(* CODESYS project Thermoversuch_00_20.project
   Description: Receives some incoming messages and echoes them with CAN-ID +1
   Company: 3S - Smart Software Solutions GmbH
   Version: 1.0.0.0
   Title: CAN Bus API Example
   Author: 3S - Smart Software Solutions GmbH

Project tree, tasks and I/O mapping:
  XLH : CODESYS Control for Raspberry Pi 64 SL, CODESYS, order no. 2302000009, version 4.12.0.0
    application app
      libraries: CAN API, 1.0.0.3 (3S - Smart Software Solutions GmbH); Standard, 3.5.18.0 (System); Memory, * (3S - Smart Software Solutions GmbH); Util, 3.5.19.0 (System); VisuDialogs, * (System); CAA Tick Extern, 3.5.17.0 (CAA Technical Workgroup); SysTime, 3.5.17.0 (System); CmpIecTask, * (System); xemax Bibliothek, 0.20 (xemax ag)
      task MAIN_TASK (cyclic, interval 20 ms, priority 0) calls MAIN, io
      task VISU_TASK (cyclic, interval 100 ms, priority 31) calls VisuElems.Visu_Prg
      program io [ST]
      Symbols
      visualisation Visualization
      program MAIN [ST]: CALL_CFC
      RNDIS_Driver
    SoftMotion General Axis Pool
    GPIOs_A_B : GPIOs B+/Pi2, CODESYS, version 4.12.0.0
        input  app.io.bSw1 : BOOL  // digital inputs (GPIO0..GPIO31).Bit4
        input  app.io.bSw2 : BOOL  // digital inputs (GPIO0..GPIO31).Bit5
        input  app.io.bSw3 : BOOL  // digital inputs (GPIO0..GPIO31).Bit6
        input  app.io.bSw4 : BOOL  // digital inputs (GPIO0..GPIO31).Bit12
        input  app.io.bSw5 : BOOL  // digital inputs (GPIO0..GPIO31).Bit13
        input  app.io.bSw6 : BOOL  // digital inputs (GPIO0..GPIO31).Bit16
        input  app.io.bSw7 : BOOL  // digital inputs (GPIO0..GPIO31).Bit17
        input  app.io.bSw8 : BOOL  // digital inputs (GPIO0..GPIO31).Bit19
        output app.io.bLed1 : BOOL  // digital outputs (GPIO0..GPIO31).Bit20
        output app.io.bLed2 : BOOL  // digital outputs (GPIO0..GPIO31).Bit21
        output app.io.bLed3 : BOOL  // digital outputs (GPIO0..GPIO31).Bit22
        output app.io.bLed4 : BOOL  // digital outputs (GPIO0..GPIO31).Bit23
        output app.io.bLed5 : BOOL  // digital outputs (GPIO0..GPIO31).Bit24
        output app.io.bLed6 : BOOL  // digital outputs (GPIO0..GPIO31).Bit26
        output app.io.bLed7 : BOOL  // digital outputs (GPIO0..GPIO31).Bit27
        unmapped channels: digital inputs (GPIO0..GPIO31), digital outputs (GPIO0..GPIO31)
    Onewire
    Camera device
      <Leer>
    SPI
    I²C
    Ethernet : Ethernet, CODESYS, version 4.2.0.0
        settings: IPAddress = [127,0,0,1]; SubnetMask = [255,0,0,0]; GatewayAddress = [0,0,0,0]; NetworkInterfaceName = 'lo'; NetworkInterfaceName = "lo"; SaveCommunicationSettings = FALSE
      ModbusTCP_Slave_OLED_Port_503 : ModbusTCP Slave Device, CODESYS, version 4.3.0.0
          settings: Port = 503
          output app.io.oled.awToOled : ARRAY[0..32] OF WORD  // Ausgänge
          unmapped channels: Eingänge
  libraries: VisuSymbols, 4.5.0.0 (System); DepictorBase, 1.0.5.0 (3S - Smart Software Solutions GmbH)
  text list GlobalTextList
  00000000-0000-0000-0000-000000000000|E:\xemax ag\prj_24_03_xLH - Allgemein\Image\RNDIS_Driver.zip
*)

// XLH/app/MAIN
PROGRAM MAIN
VAR
	bStartup: BOOL := TRUE;
	rDummy: REAL;
	bDummy: BOOL;
	data_logger: DATA_LOGGER;
	iXyDiagrammMin: INT;
	iXyDiagrammMax: INT;
	iXyDiagrammMaxVisu: INT;
	sLoggerBuffer: STRING(255);
	bRelaisVisu: BOOL;
	vVersionPlc: VERSION;
	sVersionPlc: STRING(255);
	vVersionLib: VERSION;
	sVersionLib: STRING(255);
END_VAR

// Version Bibliothex xemax
vVersionPlc.uiMajor := 0;
vVersionPlc.uiMinor := 10;
sVersionPlc := CONCAT(TO_STRING(TO_UINT(vVersionPlc.uiMajor)), CONCAT('.', (TO_STRING(TO_UINT(vVersionPlc.uiMinor)))));
vVersionLib := xemax.GetLibVersion();
sVersionLib := CONCAT(TO_STRING(TO_UINT(vVersionLib.uiMajor)), CONCAT('.', (TO_STRING(TO_UINT(vVersionLib.uiMinor)))));

IF bStartup THEN
	bStartup := FALSE;
	io.shelly.sIpShelly := '192.168.1.51';
END_IF

// Maximaler Index der Visualisierung
iXyDiagrammMax := data_logger.iIndexMax - iXyDiagrammMaxVisu;
// Status des Datenloggers
sLoggerBuffer := TO_STRING(TO_INT(MAIN.data_logger.rTimeSinceStart));
sLoggerBuffer := CONCAT(sLoggerBuffer, 's / ');
sLoggerBuffer := CONCAT(sLoggerBuffer, TO_STRING(TO_INT(data_logger.iIndexMax)));
sLoggerBuffer := CONCAT(sLoggerBuffer, 's');

bDummy := io.shelly.bRelais;
bDummy := io.shelly.bRelaisState;

rDummy := io.shelly.rVoltage;
rDummy := io.shelly.rCurrent;
rDummy := io.shelly.rActivePower;

rDummy := io.shelly.rTemperature1;
rDummy := io.shelly.rTemperature2;
rDummy := io.shelly.rTemperature3;

io.bLed1 := io.bSw1;
io.bLed2 := io.bSw2;
io.bLed3 := io.bSw3;
io.bLed4 := io.bSw4;
io.bLed5 := io.bSw5;
io.bLed6 := io.bSw6;
io.bLed7 := io.bSw7;

io.oled.bShowLines := io.bSw8;
io.oled.sLine1.sText := 'xemax ag';
io.oled.sLine2.sText := 'XLH-base';
io.oled.sLine3.sText := '';
io.oled.sLine4.sText := '';
io.oled();

CALL_CFC();

(*
Login Codesys in die XLH - SPS 
user: xlh
pw: xlh

Webvisualisierung
http://ip:8080/webvisu.htm
zBsp: http://192.168.31.31:8080/webvisu.htm

OPC-UA
anonymous (ohne Benutzer und Passwort)
opc.tcp://192.168.31.31:4840

Login XLH - Linuxumgebung via Putty
user: pi
pw: pi

Python Skript OPC-UA Autostart

crontab -e

@reboot sudo /usr/bin/python3 /home/pi/thermoversuch/thermoversuch.py


Shelly AP-Mode IP
192.168.33.1

Konfiguration WiFi 
sudo nano /etc/wpa_supplicant/wpa_supplicant.conf

network={
        ssid="xemax-xlh"
        psk="xemax-xlh"
        key_mgmt=WPA-PSK
}

mit Priorisierung
network={
   ssid="ShellyPlus1PM-C82E180598D8"
   key_mgmt=NONE
   priority=1
}


statische IP USB-Ethernet-Erweiterung: 
sudo nano /etc/dhcpcd.conf

# profile static_eth0
interface eth0
static ip_address=192.168.0.31/24

*)

ACTION CALL_CFC:
data_logger(
    rMeasureIntervall := 1.0,
    rCycleTime := xemax.TASK_INFO.rCycleTime,
    rChannel_00 := TO_REAL(io.shelly.bRelaisState),
    rChannel_01 := io.shelly.rVoltage,
    rChannel_02 := io.shelly.rCurrent,
    rChannel_03 := io.shelly.rActivePower,
    rChannel_04 := io.shelly.rApparentPower,
    rChannel_05 := io.shelly.rElectricalEnergy,
    rChannel_06 := io.shelly.rTemperatureShelly,
    rChannel_07 := io.shelly.rTemperature1,
    rChannel_08 := io.shelly.rTemperature2,
    rChannel_09 := io.shelly.rTemperature3,
    rChannel_10 := io.shelly.rTemperatureMean);
io.shelly.bResetEnergy := NOT data_logger.bEnable;
io.shelly.bRelais := bRelaisVisu OR io.bSw1;
END_ACTION

END_PROGRAM

// XLH/app/io
PROGRAM io
VAR_INPUT			
	bLed1: BOOL;
	bLed2: BOOL;
	bLed3: BOOL;
	bLed4: BOOL;
	bLed5: BOOL;
	bLed6: BOOL;
	bLed7: BOOL;	
	oled: OLED;
	shelly: SHELLY_PLUS_1PM := (rTempOffset1:=0.0, rTempOffset2:=0.0, rTempOffset3:=0.0);
END_VAR
VAR_OUTPUT
	bSw1: BOOL;
	bSw2: BOOL;
	bSw3: BOOL;
	bSw4: BOOL;
	bSw5: BOOL;
	bSw6: BOOL;
	bSw7: BOOL;
	bSw8: BOOL;
END_VAR
VAR
	bStartup: BOOL := TRUE;
END_VAR

IF bStartup THEN
	bStartup := FALSE;
END_IF

xemax.LOCAL_TIME_AND_TIME_ZONE();
xemax.TASK_INFO();
oled();
shelly(rCycleTime:=xemax.TASK_INFO.rCycleTime);

END_PROGRAM

// XLH/app/Visualization
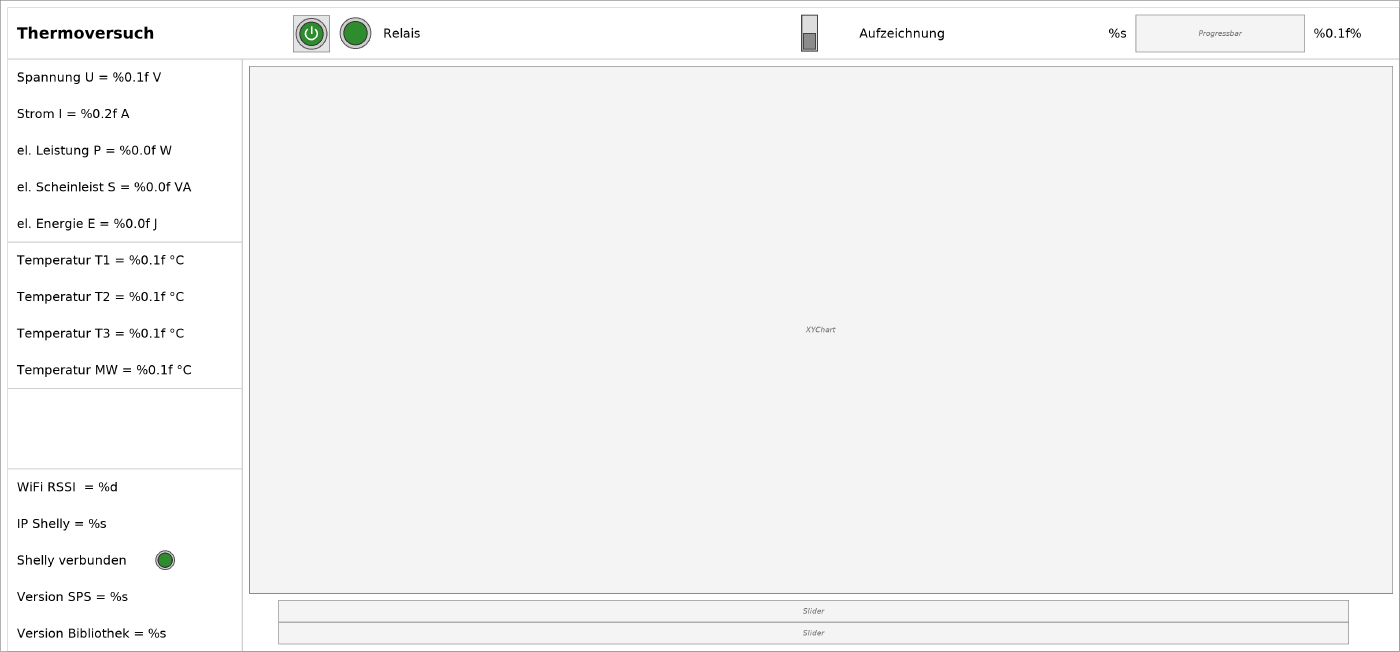
VISUALIZATION Visualization  // 1911x891
    Rectangle (10,640 321x251)
    Rectangle (10,330 321x201)
    Rectangle (330,80 1581x811)
    Rectangle (10,530 321x111)
    Rectangle (10,10 1901x71)
    Rectangle (10,80 321x251)
    PowerSwitch (400,21 50x50), variable: MAIN.bRelaisVisu, behaviour: TOGGLE, style: Switch-PowerSwitch-Green
    Rectangle (520,20 128x51), "Relais"
    Rectangle (20,20 301x51), "Thermoversuch"
    Rectangle (20,80 300x51), "Spannung U = %0.1f V", text variable: io.shelly.rVoltage
    Rectangle (20,130 300x51), "Strom I = %0.2f A", text variable: io.shelly.rCurrent
    Rectangle (20,180 300x51), "el. Leistung P = %0.0f W", text variable: io.shelly.rActivePower
    Rectangle (20,280 300x51), "el. Energie E = %0.0f J", text variable: io.shelly.rElectricalEnergy
    Rectangle (20,330 300x51), "Temperatur T1 = %0.1f °C", text variable: io.shelly.rTemperature1
    Rectangle (20,430 300x51), "Temperatur T3 = %0.1f °C", text variable: io.shelly.rTemperature3
    Rectangle (20,380 300x51), "Temperatur T2 = %0.1f °C", text variable: io.shelly.rTemperature2
    Rectangle (20,640 300x51), "WiFi RSSI = %d", text variable: io.shelly.iWiFiRssi
    Rectangle (20,480 300x51), "Temperatur MW = %0.1f °C", text variable: io.shelly.rTemperatureMean
    Line (1380,270)
    DipSwitch (1040,20 130x50), variable: MAIN.data_logger.bEnable, behaviour: TOGGLE, style: Switch-DipSwitch-Gray
    Rectangle (1170,20 141x51), "Aufzeichnung"
    Slider (380,820 1461x30), variable: MAIN.iXyDiagrammMin, scale 0..900
    Progressbar (1550,20 231x51), variable: MAIN.data_logger.rPercentFilling
    Rectangle (1790,20 111x51), "%0.1f%", text variable: MAIN.data_logger.rPercentFilling
    Rectangle (1370,20 171x51), "%s", text variable: MAIN.sLoggerBuffer
    Slider (380,850 1461x30), variable: MAIN.iXyDiagrammMaxVisu, scale 0..900
    Rectangle (20,230 300x51), "el. Scheinleist S = %0.0f VA", text variable: io.shelly.rApparentPower
    Lamp1 (460,20 50x50), variable: io.shelly.bRelaisState, style: Lamp-Lamp1-Green
    XYChart (340,90 1561x721)
    Rectangle (20,690 300x51), "IP Shelly = %s", text variable: io.shelly.sIpShelly
        OnMouseClick: write the text variable via Default
    Rectangle (20,740 221x51), "Shelly verbunden", text variable: io.shelly.sIpShelly
    Lamp1 (210,750 31x31), variable: io.shelly.bShellyConnected, style: Lamp-Lamp1-Green
    Rectangle (20,790 300x51), "Version SPS = %s", text variable: MAIN.sVersionPlc
    Rectangle (20,840 300x51), "Version Bibliothek = %s", text variable: MAIN.sVersionLib
END_VISUALIZATION
